PROGRAM MAIN
VAR
	

//runtime counter
	iCounter: INT;
	
//historize data
	fbMqttHistorize:FB_MQTT_Historize;
	
END_VAR

(*

-Test MQTT history values

*)

iCounter := iCounter +1;


fbMqttHistorize();

END_PROGRAM

(* stored: Version 1.1.0.1, ProductVersion 3.1.4024.12
   POU MAIN: Id {710da5f9-72ac-45bb-9314-a4218799ad50}, SpecialFunc None *)
